{attribute 'pack_mode' := '1'}
TYPE TMachineOptions :
STRUCT
	TurnOver		: BOOL;
	RTPearling		: BOOL;
	AutoSampling	: BOOL;
	bDisableCleanAfterPearling		: BOOL;
	bDisableVision	: BOOL;
	bSpeedModeSlow	: BOOL;
END_STRUCT
END_TYPE

(* stored: Version 1.1.0.1, ProductVersion 3.1.4022.18
   DUT TMachineOptions: Id {5384173f-523f-43b9-aae6-a73979998b13} *)
